Universal Robots PolyScope program: wrs2020_bearing_v0.urp

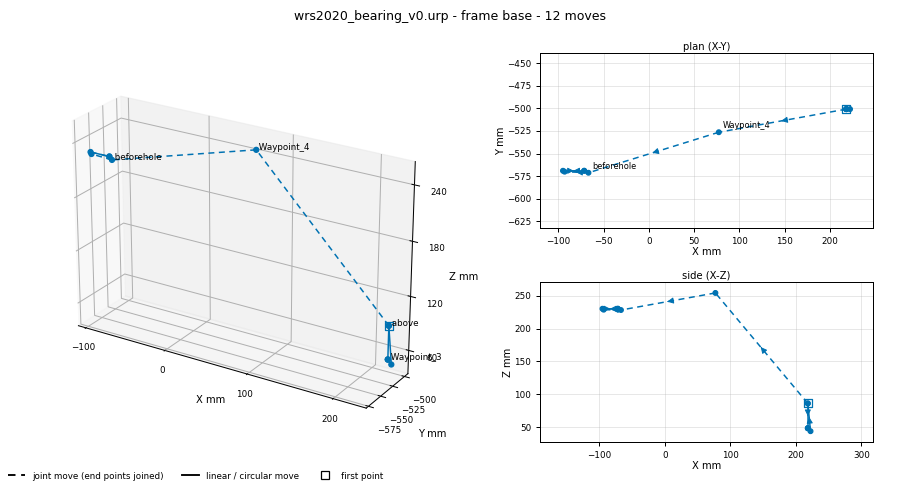
[picture p0: tool path of wrs2020_bearing_v0.urp in frame base, 12 of 16 moves have a stored position in this frame; points joined in program order, loops and branches not executed]
Program wrs2020_bearing_v0 (installation=default directory=/programs createdIn=5.7.0.90932 lastSavedIn=5.7.0.90932 robotSerialNumber=20205500607)
Calibrated DH parameters: a=[0.000096, -0.337, -0.383372, 0.000118, 0.000015, 0]; d=[0.162724, 79.377998, -95.545185, 16.300583, 0.099689, 0.099499]; alpha=[1.569249, 0.003272, 0.005201, 1.570041, -1.570219, 0]; deltaTheta=[0, 0.65664, 5.410619, 0.215927, -0.000001, 0]
Robot Program (runOnlyOnce=true)
  URCap Gripper (Robotiq_Grippers, Robotiq Inc.) dataModel(position=0.0, force=100.0, speed=100.0, positionInDouble=0.0, forceInDouble=100.0, speedInDouble=100.0, slaveIds=[9], blocking=true)
  MoveL speed 250 mm/s, acceleration 1200 mm/s^2 (useActiveTCP=true) feature=Base
    Waypoint above: TCP in base x=218.287 y=-500.902 z=86.011 mm, rx=-2.1841 ry=2.228 rz=-0.024 rad; joints [98.796, -75.562, 110.256, -124.664, -88.151, -80.024] deg; TCP offset x=0 y=0 z=165 mm, rx=0 ry=0 rz=0 rad
    Waypoint Waypoint_3: TCP in base x=218.287 y=-500.902 z=48.168 mm, rx=-2.1841 ry=2.228 rz=-0.024 rad; joints [98.784, -72.218, 112.615, -130.368, -88.157, -80] deg; TCP offset x=0 y=0 z=165 mm, rx=0 ry=0 rz=0 rad
  URCap Gripper (Robotiq_Grippers, Robotiq Inc.) dataModel(position=100.0, force=0.0, speed=0.0, positionInDouble=100.0, forceInDouble=0.0, speedInDouble=0.0, slaveIds=[9], blocking=true)
  URCap Gripper (Robotiq_Grippers, Robotiq Inc.) dataModel(position=0.0, force=0.0, speed=0.0, positionInDouble=0.0, forceInDouble=0.0, speedInDouble=0.0, slaveIds=[9], blocking=true)
  MoveL speed 600 mm/s, acceleration 1200 mm/s^2 (useActiveTCP=true) feature=Base
    Waypoint Waypoint_2: TCP in base x=218.287 y=-500.902 z=48.168 mm, rx=-0.0072 ry=3.1154 rz=0.0062 rad; joints [98.784, -72.218, 112.615, -130.368, -88.157, 8.595] deg; TCP offset x=0 y=0 z=165 mm, rx=0 ry=0 rz=0 rad
  URCap Gripper (Robotiq_Grippers, Robotiq Inc.) dataModel(position=100.0, force=0.0, speed=0.0, positionInDouble=100.0, forceInDouble=0.0, speedInDouble=0.0, slaveIds=[9], blocking=true)
  URCap Gripper (Robotiq_Grippers, Robotiq Inc.) dataModel(position=14.117647058823529, force=0.0, speed=0.0, positionInDouble=14.117647058823529, forceInDouble=0.0, speedInDouble=0.0, slaveIds=[9], blocking=true)
  MoveL speed 600 mm/s, acceleration 1200 mm/s^2 (useActiveTCP=true) feature=Base
    Waypoint Waypoint_3: TCP in base x=218.287 y=-500.902 z=48.168 mm, rx=-2.1841 ry=2.228 rz=-0.024 rad; joints [98.784, -72.218, 112.615, -130.368, -88.157, -80] deg; TCP offset x=0 y=0 z=165 mm, rx=0 ry=0 rz=0 rad
    Waypoint Waypoint_1: TCP in base x=222.423 y=-500.902 z=43.626 mm, rx=-1.9097 ry=1.9461 rz=-0.5001 rad; joints [85.342, -72.496, 119.915, -134.531, -60.23, -94.253] deg; TCP offset x=0 y=0 z=165 mm, rx=0 ry=0 rz=0 rad
  URCap Gripper (Robotiq_Grippers, Robotiq Inc.) dataModel(position=100.0, force=100.0, speed=100.0, positionInDouble=100.0, forceInDouble=100.0, speedInDouble=100.0, slaveIds=[9], blocking=true)
  MoveL speed 250 mm/s, acceleration 1200 mm/s^2 (useActiveTCP=true) feature=Base
    Waypoint above: TCP in base x=218.287 y=-500.902 z=86.011 mm, rx=-2.1841 ry=2.228 rz=-0.024 rad; joints [98.796, -75.562, 110.256, -124.664, -88.151, -80.024] deg
  SuppressedNode
    MoveJ speed 60 deg/s, acceleration 80 deg/s^2 (useActiveTCP=true) feature=Base
      Waypoint intermediate: motionParameters(blendRadius=0.05); TCP in base x=115.537 y=-464.392 z=278.491 mm, rx=2.1151 ry=-1.8246 rz=-0.1767 rad; joints [98.791, -95.537, 106.25, -108.287, -109.219, -91.027] deg
      Waypoint before_hole: TCP in base x=-57.686 y=-570.408 z=232.23 mm, rx=1.3727 ry=-1.1616 rz=-1.3181 rad; joints [97.319, -59.573, 88.654, -50.464, -171.504, -31.295] deg
  SuppressedNode
    MoveJ speed 60 deg/s, acceleration 80 deg/s^2 (useActiveTCP=true) feature=Base
      Waypoint at_hole: TCP in base x=-85.495 y=-570.408 z=232.23 mm, rx=1.3727 ry=-1.1616 rz=-1.3181 rad; joints [94.632, -61.815, 93.453, -62.169, -173.913, -40.501] deg; TCP offset x=0 y=0 z=165 mm, rx=0 ry=0 rz=0 rad
  SuppressedNode
    Force Frame feature=Joint_6_name; selection=[0, 0, 1, 0, 0, 0]; wrench=[0, 0, 10, 0, 0, 0]; limitsForce=[0.15, 0.15, 0.01, 1.047198, 1.047198, 1.047198]; limitsMotion=[0.1, 0.1, 0.1, 0.349066, 0.349066, 0.349066]
      MoveJ speed 60 deg/s, acceleration 80 deg/s^2 (useActiveTCP=true) feature=Base
        Waypoint turn_right (Relative): relativeFromPosition TCP in base x=-85.515 y=-570.41 z=232.207 mm, rx=1.3727 ry=-1.1616 rz=-1.3181 rad; joints [94.63, -61.813, 93.454, -62.171, -173.913, -40.501] deg; TCP offset x=0 y=0 z=165 mm, rx=0 ry=0 rz=0 rad; TCP in base x=-85.507 y=-570.407 z=232.241 mm, rx=0.846 ry=-1.441 rz=-0.7763 rad; joints [94.699, -63.491, 97.916, -73.842, -175.626, -8.792] deg
        Waypoint turn_left (Relative): relativeFromPosition TCP in base x=-85.52 y=-570.402 z=232.224 mm, rx=0.846 ry=-1.4411 rz=-0.7763 rad; joints [94.698, -63.49, 97.916, -73.843, -175.624, -8.792] deg; TCP in base x=-85.509 y=-570.398 z=232.173 mm, rx=1.3728 ry=-1.1615 rz=-1.3182 rad; joints [94.631, -61.811, 93.456, -62.169, -173.913, -40.501] deg
        Waypoint turn_left (Relative): relativeFromPosition TCP in base x=-85.52 y=-570.402 z=232.224 mm, rx=0.846 ry=-1.4411 rz=-0.7763 rad; joints [94.698, -63.49, 97.916, -73.843, -175.624, -8.792] deg; TCP in base x=-85.509 y=-570.398 z=232.173 mm, rx=1.3728 ry=-1.1615 rz=-1.3182 rad; joints [94.631, -61.811, 93.456, -62.169, -173.913, -40.501] deg
        Waypoint turn_right (Relative): relativeFromPosition TCP in base x=-85.515 y=-570.41 z=232.207 mm, rx=1.3727 ry=-1.1616 rz=-1.3181 rad; joints [94.63, -61.813, 93.454, -62.171, -173.913, -40.501] deg; TCP in base x=-85.507 y=-570.407 z=232.241 mm, rx=0.846 ry=-1.441 rz=-0.7763 rad; joints [94.699, -63.491, 97.916, -73.842, -175.626, -8.792] deg
  MoveJ speed 60 deg/s, acceleration 80 deg/s^2 (useActiveTCP=true) feature=Base
    Waypoint Waypoint_4: motionParameters(blendRadius=0.05); TCP in base x=77.346 y=-526.445 z=254.497 mm, rx=2.1138 ry=-1.9338 rz=-0.2706 rad; joints [93.109, -85.443, 98.102, -105.695, -107.975, -92.542] deg
    Waypoint beforehole: TCP in base x=-66.725 y=-571.237 z=228.439 mm, rx=1.497 ry=-1.6176 rz=-0.8285 rad; joints [93.116, -71.584, 102.92, -120.139, -149.991, -81.706] deg
  MoveJ speed 60 deg/s, acceleration 80 deg/s^2 (useActiveTCP=true) feature=Base
    Waypoint athole: TCP in base x=-93.062 y=-570.055 z=228.956 mm, rx=1.497 ry=-1.6176 rz=-0.8285 rad; joints [90.445, -71.97, 104.758, -126.218, -149.936, -87.03] deg
  Force Frame feature=Base; selection=[1, 0, 0, 0, 0, 0]; wrench=[-10, 0, 10, 0, 0, 0]; limitsForce=[0.01, 0.15, 0.01, 1.047198, 1.047198, 1.047198]; limitsMotion=[0.1, 0.1, 0.1, 0.349066, 0.349066, 0.349066]
    MoveL speed 50 mm/s, acceleration 200 mm/s^2 (useActiveTCP=true) feature=Base
      Waypoint rightturn (Relative): relativeFromPosition TCP in base x=-93.069 y=-570.049 z=228.937 mm, rx=1.497 ry=-1.6176 rz=-0.8285 rad; joints [90.445, -71.969, 104.759, -126.217, -149.936, -87.029] deg; TCP in base x=-93.056 y=-570.054 z=228.975 mm, rx=1.1857 ry=-1.6671 rz=-0.4357 rad; joints [90.457, -71.686, 115.038, -161.493, -150.211, -86.762] deg
      Waypoint leftturn (Relative): relativeFromPosition TCP in base x=-93.048 y=-570.049 z=228.934 mm, rx=1.1858 ry=-1.6671 rz=-0.4357 rad; joints [90.457, -71.685, 115.04, -161.493, -150.208, -86.762] deg; TCP in base x=-93.069 y=-570.047 z=228.952 mm, rx=1.497 ry=-1.6176 rz=-0.8285 rad; joints [90.445, -71.97, 104.758, -126.214, -149.936, -87.03] deg
      Waypoint leftturn (Relative): relativeFromPosition TCP in base x=-93.048 y=-570.049 z=228.934 mm, rx=1.1858 ry=-1.6671 rz=-0.4357 rad; joints [90.457, -71.685, 115.04, -161.493, -150.208, -86.762] deg; TCP in base x=-93.069 y=-570.047 z=228.952 mm, rx=1.497 ry=-1.6176 rz=-0.8285 rad; joints [90.445, -71.97, 104.758, -126.214, -149.936, -87.03] deg
      Waypoint rightturn (Relative): relativeFromPosition TCP in base x=-93.069 y=-570.049 z=228.937 mm, rx=1.497 ry=-1.6176 rz=-0.8285 rad; joints [90.445, -71.969, 104.759, -126.217, -149.936, -87.029] deg; TCP in base x=-93.056 y=-570.054 z=228.975 mm, rx=1.1857 ry=-1.6671 rz=-0.4357 rad; joints [90.457, -71.686, 115.038, -161.493, -150.211, -86.762] deg
  URCap Gripper (Robotiq_Grippers, Robotiq Inc.) dataModel(position=0.0, force=100.0, speed=100.0, positionInDouble=0.0, forceInDouble=100.0, speedInDouble=100.0, slaveIds=[9], blocking=true)
  MoveJ speed 60 deg/s, acceleration 80 deg/s^2 (useActiveTCP=true) feature=Base
    SuppressedNode
      Waypoint ready_to_push: TCP in base x=-56.908 y=-572.13 z=223.439 mm, rx=2.1027 ry=-2.324 rz=0.0706 rad; joints [70.064, -80.555, 94.786, -105.746, -87.55, -104.25] deg
    Waypoint Waypoint_6: TCP in base x=-71.45 y=-569.034 z=230.395 mm, rx=1.7826 ry=-1.97 rz=-0.6335 rad; joints [85.008, -75.761, 94.689, -108.227, -125.163, -89.082] deg
  SuppressedNode
    URCap Gripper (Robotiq_Grippers, Robotiq Inc.) dataModel(position=52.94117647058823, force=100.0, speed=100.0, positionInDouble=52.94117647058823, forceInDouble=100.0, speedInDouble=100.0, slaveIds=[9], blocking=true)
  URCap Gripper (Robotiq_Grippers, Robotiq Inc.) dataModel(position=100.0, force=100.0, speed=100.0, positionInDouble=100.0, forceInDouble=100.0, speedInDouble=100.0, slaveIds=[9], blocking=true)
  Force Frame feature=Base; selection=[1, 0, 0, 0, 0, 0]; wrench=[-100, 0, 10, 0, 0, 0]; limitsForce=[0.01, 0.15, 0.01, 1.047198, 1.047198, 1.047198]; limitsMotion=[0.1, 0.1, 0.1, 0.349066, 0.349066, 0.349066]
    MoveL speed 50 mm/s, acceleration 200 mm/s^2 (useActiveTCP=true) feature=Base
      Waypoint Waypoint_5: TCP in base x=-94.913 y=-569.034 z=230.395 mm, rx=1.7826 ry=-1.97 rz=-0.6335 rad; joints [82.679, -75.996, 95.435, -110.392, -125.156, -91.928] deg
    Wait Sleep waitTime=5
  MoveJ speed 60 deg/s, acceleration 80 deg/s^2 (useActiveTCP=true) feature=Base
    Waypoint Waypoint_6: TCP in base x=-71.45 y=-569.034 z=230.395 mm, rx=1.7826 ry=-1.97 rz=-0.6335 rad; joints [85.008, -75.761, 94.689, -108.227, -125.163, -89.082] deg
